KUKA KRL data list: service_utility.dat

&ACCESS RVO1
&REL 106
&PARAM DISKPATH = KRC:\R1\Program\CHAH
DEFDAT  service_utility PUBLIC


DECL E6POS XP1={X -231.093140,Y 607.787903,Z 875.573364,A -157.771545,B 3.09760976,C -75.8556442,S 2,T 11,E1 0.0,E2 0.0,E3 0.0,E4 0.0,E5 0.0,E6 0.0}
DECL FDAT FP1={TOOL_NO 1,BASE_NO 0,IPO_FRAME #BASE,POINT2[] " ",TQ_STATE FALSE}
DECL LDAT LCPDAT1={VEL 2.00000,ACC 100.000,APO_DIST 100.000,APO_FAC 50.0000,AXIS_VEL 100.000,AXIS_ACC 100.000,ORI_TYP #VAR,CIRC_TYP #BASE,JERK_FAC 50.0000,GEAR_JERK 50.0000,EXAX_IGN 0}
DECL E6POS XP2={X 40.6615295,Y 33.5177040,Z 689.745544,A 131.871368,B 2.79682,C 3.58198619,S 2,T 35,E1 0.0,E2 0.0,E3 0.0,E4 0.0,E5 0.0,E6 0.0}
DECL PDAT PPDAT1={VEL 100.000,ACC 100.000,APO_DIST 100.000,APO_MODE #CDIS,GEAR_JERK 50.0000,EXAX_IGN 0}

DECL PDAT PPDAT2={VEL 100.000,ACC 100.000,APO_DIST 100.000,APO_MODE #CDIS,GEAR_JERK 50.0000,EXAX_IGN 0}

DECL PDAT PPDAT3={VEL 100.000,ACC 100.000,APO_DIST 100.000,APO_MODE #CDIS,GEAR_JERK 50.0000,EXAX_IGN 0}

DECL E6POS XP6={X -587.777710,Y -1342.55969,Z 2392.72607,A 88.5205688,B -7.61228591E-13,C 180.000,S 2,T 2,E1 0.0,E2 0.0,E3 0.0,E4 0.0,E5 0.0,E6 0.0}
DECL FDAT FP6={TOOL_NO 1,BASE_NO 0,IPO_FRAME #BASE,POINT2[] " ",TQ_STATE FALSE}
DECL PDAT PPDAT5={VEL 100.000,ACC 100.000,APO_DIST 100.000,APO_MODE #CDIS,GEAR_JERK 50.0000,EXAX_IGN 0}
DECL PDAT PPDAT6={VEL 100.000,ACC 100.000,APO_DIST 100.000,APO_MODE #CDIS,GEAR_JERK 50.0000,EXAX_IGN 0}

DECL PDAT PPDAT7={VEL 100.000,ACC 100.000,APO_DIST 100.000,APO_MODE #CDIS,GEAR_JERK 50.0000,EXAX_IGN 0}

DECL PDAT PPDAT8={VEL 100.000,ACC 100.000,APO_DIST 100.000,APO_MODE #CDIS,GEAR_JERK 50.0000,EXAX_IGN 0}

DECL PDAT PPDAT9={VEL 100.000,ACC 100.000,APO_DIST 100.000,APO_MODE #CDIS,GEAR_JERK 50.0000,EXAX_IGN 0}
DECL E6POS XP10={X -112.579788,Y 522.624817,Z 379.950745,A 31.5622921,B -40.8673401,C 22.8694820,S 2,T 3,E1 0.0,E2 0.0,E3 0.0,E4 0.0,E5 0.0,E6 0.0}
DECL FDAT FP10={TOOL_NO 1,BASE_NO 0,IPO_FRAME #BASE,POINT2[] " ",TQ_STATE FALSE}
DECL PDAT PPDAT10={VEL 100.000,ACC 100.000,APO_DIST 100.000,APO_MODE #CDIS,GEAR_JERK 50.0000,EXAX_IGN 0}
DECL E6POS XP11={X -208.312927,Y 216.029419,Z 258.189453,A 44.2058868,B -0.207077980,C -37.4402733,S 2,T 3,E1 0.0,E2 0.0,E3 0.0,E4 0.0,E5 0.0,E6 0.0}
DECL FDAT FP11={TOOL_NO 1,BASE_NO 0,IPO_FRAME #BASE,POINT2[] " ",TQ_STATE FALSE}
DECL LDAT LCPDAT2={VEL 2.00000,ACC 100.000,APO_DIST 100.000,APO_FAC 50.0000,AXIS_VEL 100.000,AXIS_ACC 100.000,ORI_TYP #VAR,CIRC_TYP #BASE,JERK_FAC 50.0000,GEAR_JERK 50.0000,EXAX_IGN 0}
DECL E6POS XP12={X -226.560318,Y 234.613449,Z 292.204498,A 44.2058868,B -0.207078,C -37.4402733,S 2,T 3,E1 0.0,E2 0.0,E3 0.0,E4 0.0,E5 0.0,E6 0.0}
DECL FDAT FP12={TOOL_NO 1,BASE_NO 0,IPO_FRAME #BASE,POINT2[] " ",TQ_STATE FALSE}
DECL LDAT LCPDAT3={VEL 2.00000,ACC 100.000,APO_DIST 100.000,APO_FAC 50.0000,AXIS_VEL 100.000,AXIS_ACC 100.000,ORI_TYP #VAR,CIRC_TYP #BASE,JERK_FAC 50.0000,GEAR_JERK 50.0000,EXAX_IGN 0}
DECL E6POS XP13={X -226.560318,Y 234.613449,Z 292.204498,A -136.947189,B 1.08972490,C 37.4272232,S 2,T 35,E1 0.0,E2 0.0,E3 0.0,E4 0.0,E5 0.0,E6 0.0}
DECL FDAT FP13={TOOL_NO 1,BASE_NO 0,IPO_FRAME #BASE,POINT2[] " ",TQ_STATE FALSE}
DECL LDAT LCPDAT4={VEL 2.00000,ACC 100.000,APO_DIST 100.000,APO_FAC 50.0000,AXIS_VEL 100.000,AXIS_ACC 100.000,ORI_TYP #VAR,CIRC_TYP #BASE,JERK_FAC 50.0000,GEAR_JERK 50.0000,EXAX_IGN 0}
DECL E6POS XP14={X -193.791367,Y 201.845306,Z 188.390381,A -136.440277,B 0.689081669,C 2.31546974,S 2,T 35,E1 0.0,E2 0.0,E3 0.0,E4 0.0,E5 0.0,E6 0.0}
DECL FDAT FP14={TOOL_NO 1,BASE_NO 0,IPO_FRAME #BASE,POINT2[] " ",TQ_STATE FALSE}
DECL LDAT LCPDAT5={VEL 2.00000,ACC 100.000,APO_DIST 100.000,APO_FAC 50.0000,AXIS_VEL 100.000,AXIS_ACC 100.000,ORI_TYP #VAR,CIRC_TYP #BASE,JERK_FAC 50.0000,GEAR_JERK 50.0000,EXAX_IGN 0}
DECL E6POS XP15={X -188.422455,Y 186.762253,Z 187.951157,A -136.476929,B 0.459388047,C 0.553721368,S 2,T 35,E1 0.0,E2 0.0,E3 0.0,E4 0.0,E5 0.0,E6 0.0}
DECL FDAT FP15={TOOL_NO 1,BASE_NO 0,IPO_FRAME #BASE,POINT2[] " ",TQ_STATE FALSE}
DECL LDAT LCPDAT6={VEL 2.00000,ACC 100.000,APO_DIST 100.000,APO_FAC 50.0000,AXIS_VEL 100.000,AXIS_ACC 100.000,ORI_TYP #VAR,CIRC_TYP #BASE,JERK_FAC 50.0000,GEAR_JERK 50.0000,EXAX_IGN 0}
DECL E6POS XP16={X -290.064941,Y 288.404724,Z 187.951157,A -136.483871,B 0.543156505,C -0.0599302575,S 2,T 35,E1 0.0,E2 0.0,E3 0.0,E4 0.0,E5 0.0,E6 0.0}
DECL FDAT FP16={TOOL_NO 1,BASE_NO 0,IPO_FRAME #BASE,POINT2[] " ",TQ_STATE FALSE}
DECL LDAT LCPDAT7={VEL 2.00000,ACC 100.000,APO_DIST 100.000,APO_FAC 50.0000,AXIS_VEL 100.000,AXIS_ACC 100.000,ORI_TYP #VAR,CIRC_TYP #BASE,JERK_FAC 50.0000,GEAR_JERK 50.0000,EXAX_IGN 0}
DECL PDAT PPDAT11={VEL 100.000,ACC 100.000,APO_DIST 100.000,APO_MODE #CDIS,GEAR_JERK 50.0000,EXAX_IGN 0}
DECL PDAT PPDAT12={VEL 100.000,ACC 100.000,APO_DIST 100.000,APO_MODE #CDIS,GEAR_JERK 50.0000,EXAX_IGN 0}
DECL PDAT PPDAT13={VEL 100.000,ACC 100.000,APO_DIST 100.000,APO_MODE #CDIS,GEAR_JERK 50.0000,EXAX_IGN 0}
DECL BASIS_SUGG_T LAST_BASIS={POINT1[] "P0                      ",POINT2[] "P0                      ",CP_PARAMS[] "CPDAT0                  ",PTP_PARAMS[] "PDAT0                   ",CONT[] "                        ",CP_VEL[] "2.0                     ",PTP_VEL[] " 100                    ",SYNC_PARAMS[] "SYNCDAT                 ",SPL_NAME[] "S0                      ",A_PARAMS[] "ADAT0                   "}
DECL E6POS XPICK_POINT={X 230.048477,Y 1.62400365,Z -0.623077810,A 179.392990,B 1.62171900,C 179.904175,S 2,T 34,E1 0.0,E2 0.0,E3 0.0,E4 0.0,E5 0.0,E6 0.0}
DECL FDAT Fpick_point={TOOL_NO 0,BASE_NO 1,IPO_FRAME #BASE,POINT2[] " ",TQ_STATE FALSE}
DECL LDAT LCPDAT8={VEL 2.00000,ACC 100.000,APO_DIST 100.000,APO_FAC 50.0000,AXIS_VEL 100.000,AXIS_ACC 100.000,ORI_TYP #VAR,CIRC_TYP #BASE,JERK_FAC 50.0000,GEAR_JERK 50.0000,EXAX_IGN 0}
DECL TQM_TQDAT_T TM1={T11 3,T12 12,T13 3,T14 0,T15 4,T16 2,T21 44801,T22 84472,T23 44002,T24 0,T25 25580,T26 8826,K1 301,K2 299,K3 300,K4 0,K5 300,K6 297,O1 20,O2 30,ID 1,OVM 100,TMF 1.00000}

DECL E6POS XPP_OVER={X 358.468750,Y 95.9617233,Z 27.9932518,A 0.379252136,B -1.10826421,C -0.375179052,S 2,T 43,E1 0.0,E2 0.0,E3 0.0,E4 0.0,E5 0.0,E6 0.0}
DECL FDAT Fpp_over={TOOL_NO 1,BASE_NO 1,IPO_FRAME #BASE,POINT2[] " ",TQ_STATE FALSE}
DECL PDAT PPDAT14={VEL 100.000,ACC 100.000,APO_DIST 100.000,APO_MODE #CDIS,GEAR_JERK 50.0000,EXAX_IGN 0}
DECL TQM_TQDAT_T TM2={T11 14,T12 10,T13 6,T14 0,T15 6,T16 14,T21 234438,T22 106507,T23 152141,T24 0,T25 41095,T26 30205,K1 301,K2 299,K3 300,K4 0,K5 300,K6 297,O1 20,O2 30,ID 2,OVM 100,TMF 1.00000}
DECL LDAT LCPDAT9={VEL 2.00000,ACC 100.000,APO_DIST 100.000,APO_FAC 50.0000,AXIS_VEL 100.000,AXIS_ACC 100.000,ORI_TYP #VAR,CIRC_TYP #BASE,JERK_FAC 50.0000,GEAR_JERK 50.0000,EXAX_IGN 0}
DECL LDAT LCPDAT10={VEL 2.00000,ACC 100.000,APO_DIST 100.000,APO_FAC 50.0000,AXIS_VEL 100.000,AXIS_ACC 100.000,ORI_TYP #VAR,CIRC_TYP #BASE,JERK_FAC 50.0000,GEAR_JERK 50.0000,EXAX_IGN 0}
DECL E6POS XPRE_PP={X 109.612343,Y 143.284927,Z -1036.37244,A 90.0611572,B 0.00371537823,C 179.891907,S 2,T 10,E1 0.0,E2 0.0,E3 0.0,E4 0.0,E5 0.0,E6 0.0}
DECL FDAT Fpre_pp={TOOL_NO 0,BASE_NO 1,IPO_FRAME #BASE,POINT2[] " ",TQ_STATE FALSE}
DECL PDAT PPDAT4={VEL 100.000,ACC 100.000,APO_DIST 100.000,APO_MODE #CDIS,GEAR_JERK 50.0000,EXAX_IGN 0}
DECL LDAT LCPDAT0={VEL 2.00000,ACC 100.000,APO_DIST 100.000,APO_FAC 50.0000,AXIS_VEL 100.000,AXIS_ACC 100.000,ORI_TYP #VAR,CIRC_TYP #BASE,JERK_FAC 50.0000,GEAR_JERK 50.0000,EXAX_IGN 0}
DECL E6POS XCENTER={X 1932.57556,Y 8.92797947,Z 2065.98682,A 179.999725,B -6.88975244E-14,C -180.000,S 2,T 43,E1 0.0,E2 0.0,E3 0.0,E4 0.0,E5 0.0,E6 0.0}
DECL AXIS ACENTER={A2 -110.000,A3 86.0000}
DECL FDAT Fcenter={TOOL_NO 0,BASE_NO 0,IPO_FRAME #BASE,POINT2[] " ",TQ_STATE FALSE}
DECL PDAT PPDAT15={VEL 100.000,ACC 100.000,APO_DIST 100.000,APO_MODE #CDIS,GEAR_JERK 50.0000,EXAX_IGN 0}
DECL PDAT PPDAT16={VEL 100.000,ACC 100.000,APO_DIST 400.000,APO_MODE #CDIS,GEAR_JERK 50.0000,EXAX_IGN 0}
DECL E6POS XPICK_POINT_2={X 242.124924,Y 4.23651934,Z -19.2544823,A -179.899780,B 1.60807776,C -179.245438,S 2,T 11,E1 0.0,E2 0.0,E3 0.0,E4 0.0,E5 0.0,E6 0.0}
DECL FDAT Fpick_point_2={TOOL_NO 0,BASE_NO 2,IPO_FRAME #BASE,POINT2[] " ",TQ_STATE FALSE}
DECL LDAT LCPDAT11={VEL 2.00000,ACC 100.000,APO_DIST 100.000,APO_FAC 50.0000,AXIS_VEL 100.000,AXIS_ACC 100.000,ORI_TYP #VAR,CIRC_TYP #BASE,JERK_FAC 50.0000,GEAR_JERK 50.0000,EXAX_IGN 0}
DECL E6POS XPICK_POINT_3={X -533.826233,Y -1174.06030,Z 2962.14941,A 89.8363342,B 1.74666495E-14,C -180.000,S 2,T 2,E1 0.0,E2 0.0,E3 0.0,E4 0.0,E5 0.0,E6 0.0}
DECL FDAT Fpick_point_3={TOOL_NO 1,BASE_NO 0,IPO_FRAME #BASE,POINT2[] " ",TQ_STATE FALSE}
DECL PDAT PPDAT17={VEL 100.000,ACC 100.000,APO_DIST 100.000,APO_MODE #CDIS,GEAR_JERK 50.0000,EXAX_IGN 0}
DECL E6POS Xserv={X -533.826233,Y -1174.06030,Z 2962.14941,A 89.8363342,B 1.74666495E-14,C -180.000,S 2,T 2,E1 0.0,E2 0.0,E3 0.0,E4 0.0,E5 0.0,E6 0.0}
DECL FDAT Fserv={TOOL_NO 1,BASE_NO 0,IPO_FRAME #BASE,POINT2[] " ",TQ_STATE FALSE}
ENDDAT
